// TIA Portal V17 export
// export: Created 2025-03-07T09:24:20.4035684Z, ExportSetting WithDefaults, DisplayName Totally Integrated Automation Portal, DisplayVersion V17 Update 8, DisplayName TIA Portal Openness, DisplayVersion V17 Update 8, DisplayName TIA Portal Version Control Interface, DisplayVersion V17, DisplayName SINAMICS Startdrive Advanced, DisplayVersion V17 SP2, DisplayName SINAMICS Startdrive G110M, G120, G120C, G120D, G120P, G115D, DisplayVersion V17 SP2, DisplayName SINAMICS Startdrive G130, G150, S120, S150, SINAMICS MV, S210, DisplayVersion V17 SP2, DisplayName STEP 7 Professional, DisplayVersion V17 Update 8, DisplayName SINUMERIK ONE STEP 7 Toolbox, DisplayVersion V17 Update 12, DisplayName SINUMERIK 840D sl STEP 7 Toolbox, DisplayVersion V17 Update 12, DisplayName STEP 7 Safety, DisplayVersion V17 Update 6, DisplayName WinCC Advanced, DisplayVersion V17 Update 8
DATA_BLOCK "DB22332_PRESSURIZE_GAS_VALVE_HOPPER_2_UNIT_02"   // DB22332
{ DB_Accessible_From_OPC_UA := 'FALSE' }
VERSION : 0.1
// stored: AutoNumber false, DBAccessibleFromOPCUA false, DBAccessibleFromWebserver true, InstanceOfName FB22301_SOLENOID_VALVE, InstanceOfType FB
"FB22301_SOLENOID_VALVE"
   // VAR_INPUT
   //    iCONTROL_ON_DELAYED : Bool;
   //    iPNEUMATIC_FEEDBACK_ON : Bool;
   //    iMANUAL_START_REQUEST : Bool;
   //    iAUTO_START_REQUEST : Bool;
   //    iMANUAL_STOP_REQUEST : Bool;
   //    iAUTO_STOP_REQUEST : Bool;
   // END_VAR
   // VAR_OUTPUT
   //    oSYSTEM_ON : Bool;
   // END_VAR
   // VAR RETAIN
   //    "DATA STANDARD" { S7_SetPoint := 'True'} : "GENERAL_DATA_START_STOP";
   //    "HMI STANDARD" { S7_SetPoint := 'True'} : "HMI_DATA_START_STOP";
   // END_VAR
BEGIN
END_DATA_BLOCK
